FUNCTION_BLOCK MainAppGUIFB (* JADE WORKER *)
  (* Standard: 61499-1 *)
  (* Version 1.0, 2014-04-22, Ahmed, Fraunhofer IGD *)
  (* Compiler header: package fb.rt; *)
  (* Compiler Java Sun JDK 1.5.0 *)
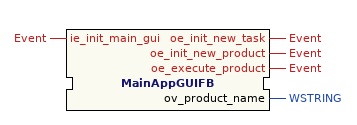
  EVENT_INPUT
    ie_init_main_gui;
  END_EVENT
  EVENT_OUTPUT
    oe_init_new_task;
    oe_init_new_product;
    oe_execute_product;
  END_EVENT
  VAR_OUTPUT
    ov_product_name : WSTRING;
  END_VAR
END_FUNCTION_BLOCK
